(* PLC project Blank Project, Blank Blank 1.0 *)
(* stored: creationDateTime 2016-05-18T21:14:07, modificationDateTime 2021-04-13T12:00:53 *)

PROGRAM CB_failure_Prot
  VAR
    CB_FDR1_failure : BOOL;
    CB_FDR4_failure : BOOL;
    CB1_22KV_failure : BOOL;
    CB3_22KV_failure : BOOL;
  END_VAR
  VAR
    Open_CB1_22KV AT %QX0.0 : BOOL;
    Open_CB2_22KV AT %QX0.1 : BOOL;
    Open_CB3_22KV AT %QX0.2 : BOOL;
    Open_CB_TRSF1 AT %QX0.3 : BOOL;
    Open_CB_TRSF2 AT %QX0.4 : BOOL;
    Reset_All_CB AT %IX0.0 : BOOL;
    Status_CB1_22KV AT %IX0.1 : BOOL;
    Status_CB3_22KV AT %IX0.2 : BOOL;
    Status_CB_FDR1 AT %IX0.3 : BOOL;
    Status_CB_FDR4 AT %IX0.4 : BOOL;
    Fault_on_FDR1_Current AT %IW0 : INT;
    Fault_on_FDR4_Current AT %IW1 : INT;
    Fault_on_22BUS1_Current AT %IW2 : INT;
    Fault_on_22BUS2_Current AT %IW3 : INT;
  END_VAR
  VAR
    Threshold500 : INT := 500;
    TON0 : TON;
    TON1 : TON;
    TON2 : TON;
    TON3 : TON;
  END_VAR

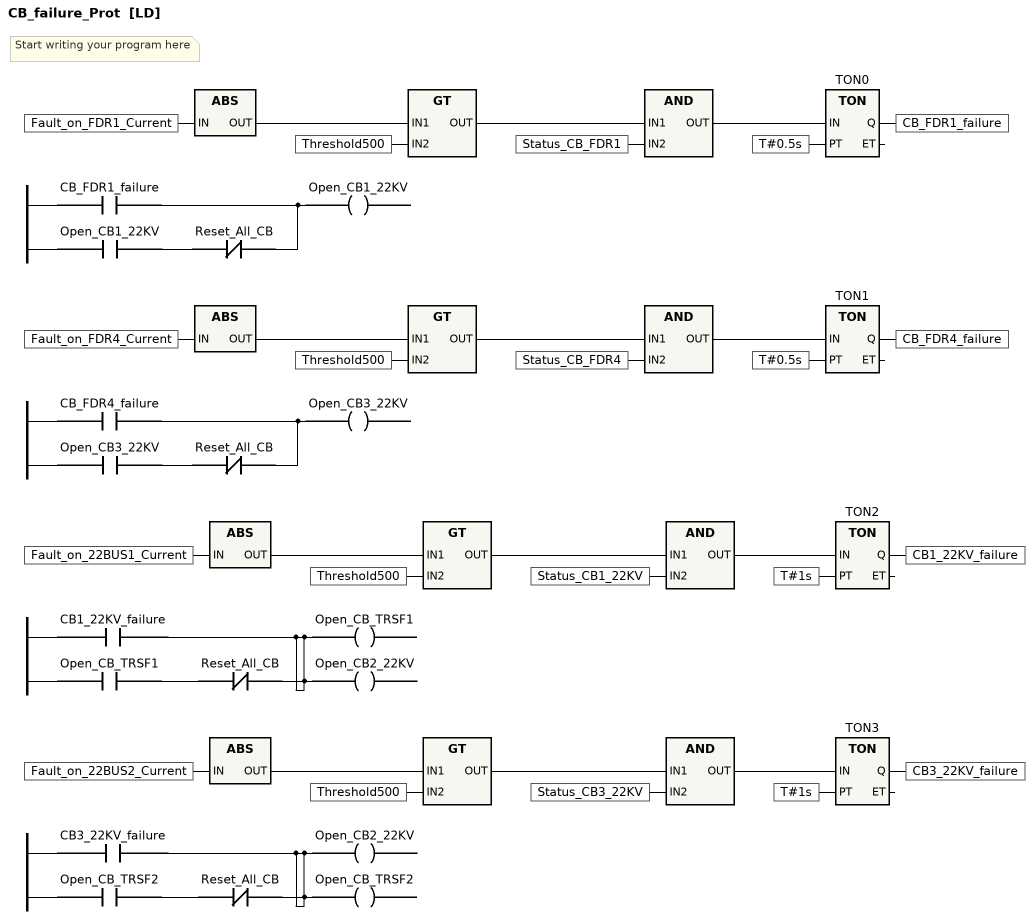
(* LD diagram, written out as Structured Text *)
(* Start writing your program here *)
Open_CB1_22KV := CB_FDR1_failure OR Open_CB1_22KV AND NOT Reset_All_CB;
TON0(IN := ABS(Fault_on_FDR1_Current) > Threshold500 AND Status_CB_FDR1, PT := T#0.5s);
CB_FDR1_failure := TON0.Q;
Open_CB3_22KV := CB_FDR4_failure OR Open_CB3_22KV AND NOT Reset_All_CB;
TON1(IN := ABS(Fault_on_FDR4_Current) > Threshold500 AND Status_CB_FDR4, PT := T#0.5s);
CB_FDR4_failure := TON1.Q;
Open_CB2_22KV := CB1_22KV_failure OR Open_CB_TRSF1 AND NOT Reset_All_CB;
Open_CB_TRSF1 := CB1_22KV_failure OR Open_CB_TRSF1 AND NOT Reset_All_CB;
TON2(IN := ABS(Fault_on_22BUS1_Current) > Threshold500 AND Status_CB1_22KV, PT := T#1s);
CB1_22KV_failure := TON2.Q;
Open_CB2_22KV := CB3_22KV_failure OR Open_CB_TRSF2 AND NOT Reset_All_CB;
Open_CB_TRSF2 := CB3_22KV_failure OR Open_CB_TRSF2 AND NOT Reset_All_CB;
TON3(IN := ABS(Fault_on_22BUS2_Current) > Threshold500 AND Status_CB3_22KV, PT := T#1s);
CB3_22KV_failure := TON3.Q;
END_PROGRAM

CONFIGURATION Config0
  RESOURCE Res0 ON PLC
    TASK TaskMain(INTERVAL := T#10ms, PRIORITY := 0);
    PROGRAM Inst0 WITH TaskMain : CB_failure_Prot;
  END_RESOURCE
END_CONFIGURATION
